// SIMATIC S7-200 project (STEP 7-Micro/WIN), CPU 221 REL 01.10

ORGANIZATION_BLOCK 主程序:OB1
TITLE=程序注释
BEGIN
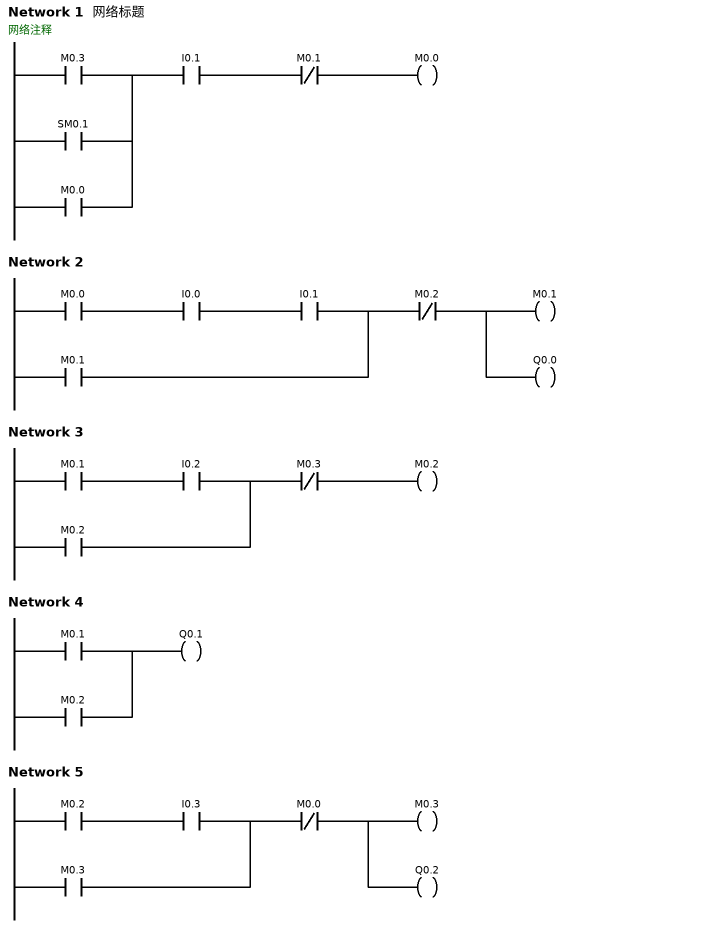
Network 1 // 网络标题
// 网络注释
LD     M0.3
O      SM0.1
O      M0.0
A      I0.1
AN     M0.1
=      M0.0
Network 2
LD     M0.0
A      I0.0
A      I0.1
O      M0.1
AN     M0.2
=      M0.1
=      Q0.0
Network 3
LD     M0.1
A      I0.2
O      M0.2
AN     M0.3
=      M0.2
Network 4
LD     M0.1
O      M0.2
=      Q0.1
Network 5
LD     M0.2
A      I0.3
O      M0.3
AN     M0.0
=      M0.3
=      Q0.2
END_ORGANIZATION_BLOCK
